FUNCTION_BLOCK CONSOLE (* Output Qualified Event+Data to Console *)
  (* Standard: 61499-2 *)
  (* Version 0.0, 2000-04-03, JHC, Rockwell Automation *)
  (* Compiler header: package fb.rt.hmi; *)
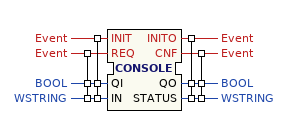
  EVENT_INPUT
    INIT WITH QI, IN; (* Initialization Event *)
    REQ WITH QI, IN; (* Request Event *)
  END_EVENT
  EVENT_OUTPUT
    INITO WITH QO, STATUS; (* Initialization Confirm *)
    CNF WITH QO, STATUS; (* Output Confirm *)
  END_EVENT
  VAR_INPUT
    QI : BOOL;
    IN : WSTRING;
  END_VAR
  VAR_OUTPUT
    QO : BOOL; (* Copy of QI *)
    STATUS : WSTRING; (* Copy of IN *)
  END_VAR
END_FUNCTION_BLOCK
